FUNCTION_BLOCK PUBLIC FB_SequenceSortedByDurationDescending IMPLEMENTS I_SequenceSortable
VAR_INPUT
END_VAR
VAR_OUTPUT
END_VAR
VAR
END_VAR

METHOD SortList
VAR_INPUT
	refSequence			: REFERENCE TO ARRAY [1..5] OF ST_SequenceItem;
END_VAR
VAR
	stLeft, stRight		: ST_SequenceItem;
	nMax, nIndex		: INT;
	bSwapped			: BOOL;
END_VAR
REPEAT
	bSwapped := FALSE;
	FOR nIndex := 1 TO 4 DO
		stLeft := refSequence[nIndex];
		stRight := refSequence[nIndex + 1];
		IF (stLeft.nDuration < stRight.nDuration) THEN
			refSequence[nIndex + 1] := stLeft;
			refSequence[nIndex] := stRight;
			bSwapped := TRUE;
		END_IF
	END_FOR
UNTIL
	bSwapped = FALSE
END_REPEAT;
END_METHOD

END_FUNCTION_BLOCK

(* stored: Version 1.1.0.1, ProductVersion 3.1.4024.12
   POU FB_SequenceSortedByDurationDescending: Id {8408adc7-ad39-439f-961d-7db169bcf9b6}, SpecialFunc None
   Method SortList: Id {5eefbf68-aec6-4ff1-82ea-389279877599} *)
